{attribute addProperty BoxType "EL2911-0000-0016"}
{attribute addProperty Id "Standard_OutputAT %Q*BOOL81"}
{attribute addProperty CRC "3131824585"}
{attribute addProperty SizeInBites "8"}
{attribute addProperty SizeInBytes "1"}
TYPE Outputs_BAABD9C9 :
STRUCT
	{attribute addProperty Name "Standard_Output"}
	Standard_Output AT %Q* : BOOL;
END_STRUCT
END_TYPE

(* stored: Version 1.2.0.0, ProductVersion 3.1.4024.9
   DUT Outputs_BAABD9C9: Id {8d65f01d-cd85-478c-8528-96fda3eec5a5} *)
